// TIA Portal V19 export
TYPE "LEXCHANGETRAY_typeRollerVfdContronNode"
// commandConfiguration: LEXCHANGETRAY_typeRollerVfdContronNodeCommandConfiguration
// commands: LEXCHANGETRAY_typeRollerVfdContronNodeCommands
// monitoring: LEXCHANGETRAY_typeVfdContronNodeMonitoring
// stored: Access Published
   STRUCT
      commandConfiguration { S7_SetPoint := 'True'} : "LEXCHANGETRAY_typeRollerVfdContronNodeCommandConfiguration";
      commands { S7_SetPoint := 'True'} : "LEXCHANGETRAY_typeRollerVfdContronNodeCommands";
      monitoring { S7_SetPoint := 'True'} : "LEXCHANGETRAY_typeVfdContronNodeMonitoring";
   END_STRUCT;
END_TYPE
